(*
SPDX-FileCopyrightText: © 2026 Oleksandr Tiutyk <trofimich@gmail.com>
SPDX-License-Identifier: MIT
License: https://opensource.org/license/mit
*)

{attribute 'qualified_only'}
{attribute 'strict'}
{attribute 'to_string'}
TYPE DIRECTION_TYPE :
(
	NEGATIVE := -1,
	UNDEFINED := 0,
	POSITIVE := 1
) SINT;
END_TYPE

(* stored: Version 1.1.0.1
   DUT DIRECTION_TYPE: Id {37edcb9d-b405-4b92-939a-8037a23e260d} *)
